// Exemple illustrates how to iterate thru Objectlists to query statusflags
FUNCTION_BLOCK FB_BACnet_StatusFlags 
VAR_INPUT
	bEnPolling				: BOOL;	
	bIterate				: BOOL; 
END_VAR
VAR_OUTPUT
	nInAlarm				: DINT;
	nFault					: DINT;
	nOverridden				: DINT;
	nOutOfService			: DINT;	 
END_VAR
VAR
	{region 'Iteration'}
	// Intention:			Iterate over Objectlist.
	bDebugMsg				: BOOL;	
	bIterate_ShowObjects	: BOOL				:= FALSE;	 
	bIterate_ShowObjectType	: BOOL				:= TRUE;
	bIterate_ShowFlags		: BOOL				:= TRUE;			 
			 
	{endregion}

	tonPolling				: Ton:=(PT:=T#5S) ;
END_VAR
VAR	

	ST_StateFlags			: ST_BA_StatusFlags;	
	_i						: DINT;
	_sVal					: T_MaxString;
	_iObj					: I_BA_Object;
	_iEvtObj				: I_BA_EventObject;
	_fbMsg					: FB_BA_DecorString;
END_VAR

IF bEnPolling THEN
	bDebugMsg:=FALSE;
	tonPolling.IN:=NOT tonPolling.Q;
	tonPolling();
ELSE	
	tonPolling.IN:=FALSE;
END_IF 


IF (bIterate)or (tonPolling.Q) THEN
	bIterate := FALSE;
	
	IF (bDebugMsg) THEN	
		_i := F_BA_GetEventCount();
		IF (_i = 0) THEN
			F_BA_LogMessage(ADSLOG_MSGTYPE_HINT, 'EM06', 'No active events found yet.');
		ELSE
			F_BA_LogMessage1(ADSLOG_MSGTYPE_HINT, 'EM08', 'Active events: %d', F_DINT(_i));
		END_IF
	END_IF
		// Iterate over all active events:
		nOverridden:=0;
		nOutOfService:=0;
		nInAlarm:=0;
		nFault:=0;
		_i := 0;
		_iObj := 0;								// [Hint] Temporary iterator-object must be NULL to start iteration from the beginning.
		WHILE (F_BA_IterateObjects(_iObj)) DO
			_i := (_i+1);			
        
			IF (__QUERYINTERFACE(_iObj,_iEvtObj))	THEN
				IF 	_iEvtObj.ObjectType = E_BA_Objecttype.eStructuredView THEN
					;
				ELSE
				// Format message:
					_fbMsg.Reset();
					
					IF (bIterate_ShowObjectType) THEN
						_sVal := TO_STRING(_iEvtObj.ObjectType);
						_fbMsg.AddDecor1('ObjectType: %s', F_STRING(_sVal));
					END_IF
					// Read Flags
					IF (bIterate_ShowFlags) THEN						
						ST_StateFlags:= _iEvtObj.StateFlags;
						_sVal := TO_STRING(F_BA_StatusFlags_ToRaw(stValue:=ST_StateFlags ));
						_fbMsg.AddDecor1('Flags: %s', F_STRING(_sVal));
						IF ST_StateFlags.bOverridden THEN
								nOverridden:=nOverridden+1;
						END_IF
						IF ST_StateFlags.bOutOfService THEN
								nOutOfService:=nOutOfService+1;
						END_IF
						IF ST_StateFlags.bFault THEN
								nFault:=nFault+1;
						END_IF
						IF ST_StateFlags.bInAlarm THEN
								nInAlarm:=nInAlarm+1;
						END_IF
					END_IF
					
					_fbMsg.Finish();
					
					IF (bIterate_ShowObjects) THEN						
						_sVal := _iObj.ObjectName;
						F_BA_LogMessage3(ADSLOG_MSGTYPE_HINT, 'EM32', '%d. %s   %s', F_DINT(_i), F_STRING(_sVal), F_STRING(_fbMsg.sOutput));
					END_IF
				END_IF
			
			END_IF
        
			END_WHILE
			IF (bDebugMsg) THEN	
				F_BA_LogMessage1(ADSLOG_MSGTYPE_HINT, 'EM10', 'Objects InAlarm: %d', F_DINT(nInAlarm));
				F_BA_LogMessage1(ADSLOG_MSGTYPE_HINT, 'EM11', 'Objects Fault: %d', F_DINT(nFault));
				F_BA_LogMessage1(ADSLOG_MSGTYPE_HINT, 'EM12', 'Objects Overridden: %d', F_DINT(nOverridden));
				F_BA_LogMessage1(ADSLOG_MSGTYPE_HINT, 'EM13', 'Objects OutOfService: %d', F_DINT(nOutOfService));
			END_IF
				
END_IF

END_FUNCTION_BLOCK

(* stored: Version 1.1.0.1, ProductVersion 3.1.4024.12
   POU FB_BACnet_StatusFlags: Id {d450a52c-a6c9-44d0-91bf-a7d196a6032a}, SpecialFunc None *)
